// TIA Portal project "hamiev1" (V15)

(* hardware
DEVICE "S7-1200 station_1"  S7-1200 Station
   slot 0: "Rack_0"  S7-1200 Rack  Rack  V1.0
   slot 1: "PLC_1"  CPU 1214C DC/DC/Rly  6ES7 214-1HG40-0XB0  V4.2
*)

// ===== PLC "PLC_1"  CPU 1214C DC/DC/Rly =====

VAR_GLOBAL   // PLC tag table "Default tag table"
   "start" AT %M0.0 : Bool;
   "stop" AT %M0.1 : Bool;
   "pump1" AT %Q0.3 : Bool;
   "lowsensor" AT %M0.3 : Bool;
   "highsensor" AT %M0.4 : Bool;
   "motor" AT %Q0.1 : Bool;
   "pump3" AT %Q0.2 : Bool;
   "Tag_1" AT %M1.1 : Bool;
   "active" AT %M0.2 : Bool;
   "tg1" AT %M0.5 : Bool;
END_VAR

// folder: System blocks/Program resources

DATA_BLOCK "IEC_Timer_0_DB"   // DB1
{ S7_Optimized_Access := 'TRUE' }
AUTHOR : Simatic
FAMILY : IEC
NAME : IEC_TMR
VERSION : 1.0
// stored: InstanceOfName IEC_TIMER
"IEC_TIMER"
BEGIN
END_DATA_BLOCK

// folder: (top level)

ORGANIZATION_BLOCK "Main"   // OB1, LAD, ProgramCycle
TITLE = "Main Program Sweep (Cycle)"
{ S7_Optimized_Access := 'TRUE' }
VERSION : 0.1
   VAR_INPUT
      Initial_Call : Bool;   // Initial call of this OB
      Remanence : Bool;   // =True, if remanent data are available
   END_VAR
   VAR_TEMP   // added for the SCL form of the ladder/FBD networks
      _w1 : Bool;
   END_VAR
BEGIN

REGION Network 1
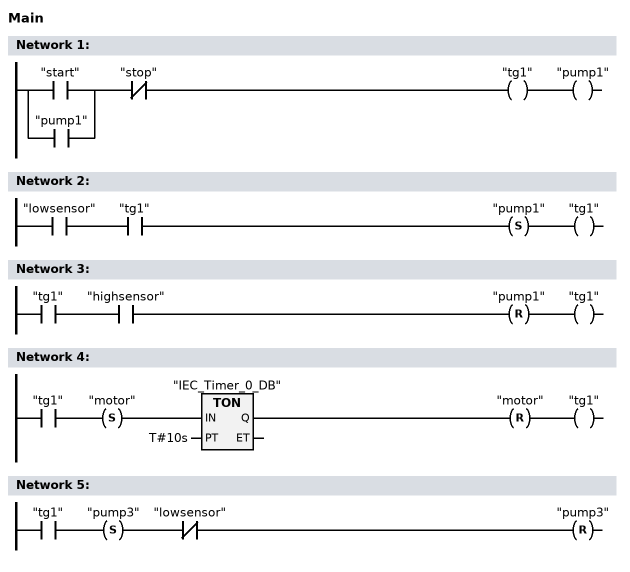
   RUNG wire#powerrail
      Contact( "start" )
      wire#w1
      I_Contact( "stop" )
      Coil( "tg1" )
      Coil( "pump1" )
   END_RUNG
   RUNG wire#powerrail
      Contact( "pump1" )
   END_RUNG wire#w1
   // the same network as SCL:
   "tg1" := ("start" OR "pump1") AND NOT "stop";
   "pump1" := "tg1";
END_REGION

REGION Network 2
   RUNG wire#powerrail
      Contact( "lowsensor" )
      Contact( "tg1" )
      S_Coil( "pump1" )
      Coil( "tg1" )
   END_RUNG
   // the same network as SCL:
   #_w1 := "lowsensor" AND "tg1";
   IF #_w1 THEN "pump1" := TRUE; END_IF;
   "tg1" := #_w1;
END_REGION

REGION Network 3
   RUNG wire#powerrail
      Contact( "tg1" )
      Contact( "highsensor" )
      R_Coil( "pump1" )
      Coil( "tg1" )
   END_RUNG
   // the same network as SCL:
   #_w1 := "tg1" AND "highsensor";
   IF #_w1 THEN "pump1" := FALSE; END_IF;
   "tg1" := #_w1;
END_REGION

REGION Network 4
   IF "tg1" THEN "motor" := TRUE; END_IF;
   "IEC_Timer_0_DB".TON(IN := "tg1", PT := T#10s);
   IF "IEC_Timer_0_DB".Q THEN "motor" := FALSE; END_IF;
   "tg1" := "IEC_Timer_0_DB".Q;
END_REGION

REGION Network 5
   RUNG wire#powerrail
      Contact( "tg1" )
      S_Coil( "pump3" )
      I_Contact( "lowsensor" )
      R_Coil( "pump3" )
   END_RUNG
   // the same network as SCL:
   IF "tg1" THEN "pump3" := TRUE; END_IF;
   IF "tg1" AND NOT "lowsensor" THEN "pump3" := FALSE; END_IF;
END_REGION
END_ORGANIZATION_BLOCK